// Mitsubishi GX Works2 project: Group27   PLC: FX3G

// global labels: Global1
VAR_GLOBAL
  Start_Day AT X007 : BOOL;
  Input_Raspberry AT D1100 : INT;
  Raspberry AT D1200 : INT;
  Input_Lemon AT D1300 : INT;
  Lemon AT D1400 : INT;
  Input_Stabilizer AT D1500 : INT;
  Stabilizer AT D1600 : INT;
  Input_Gummybears AT D1700 : INT;
  Gummybears AT D1800 : INT;
  Analog_Output2 AT D2500 : INT;
  Choice AT D1900 : REAL;
  Raspberry_Icecream_Container AT D2000 : INT;
  Lemon_Icecream_Cointainer AT D2100 : INT;
  Analog_Input1 AT D8280 : INT;
  Raspberry_Icecream_Cooler AT D2200 : INT;
  Lemon_Icecream_Cooler AT D2300 : INT;
  Mixing_Container AT D2400 : INT;
  Not_Enough_Material AT M1 : BOOL;
  Normal_Lamp AT M2 : BOOL;
  Pinuk_Lamp AT M3 : BOOL;
  Finished_Move_Cool AT M4 : BOOL;
  Cool_Finished AT M5 : BOOL;
  Trigger_Blink AT M6 : BOOL;
  Finish_Work AT M7 : BOOL;
  Zero AT K0 : INT;
  In_Work AT Y007 : BOOL;
  Emergency_Switch AT X005 : BOOL;
  Sample AT X001 : BOOL;
  Analog_Output AT D8282 : INT;
  Divider_400 AT E400 : REAL;
  Max_Normal AT E5 : REAL;
  Min_Pinuk AT E5 : REAL;
  Min_Raspberry_Normal AT K280 : INT;
  Min_Raspberry_Pinuk AT K385 : INT;
  Min_Lemon_Normal AT K455 : INT;
  Min_Lemon_Pinuk AT K665 : INT;
  Min_Stabilizer_Normal AT K105 : INT;
  Min_Stabilizer_Pinuk AT K210 : INT;
  Min_Gummybear_Normal AT K28 : INT;
  Min_Gummybear_Pinuk AT K70 : INT;
  Raspberry_Icecream_Normal AT K350 : INT;
  Raspberry_Icecream_Pinuk AT K560 : INT;
  Lemon_Icecream_Normal AT K490 : INT;
  Lemon_Icecream_Pinuk AT K700 : INT;
  Add_Pack AT K1 : INT;
  One_Sec AT K10 : INT;
  Three_Sec AT K30 : INT;
  Five_Sec AT K50 : INT;
  Eight_Sec AT K80 : INT;
  Normal_Icecram AT K868 : INT;
  Pinuk_Icecram AT K1330 : INT;
  Multiply_40 AT K40 : INT;
  First_Step_Timer AT TC0 : BOOL;
  Step1_Finished AT TS0 : BOOL;
  Icecream_Making AT Y000 : BOOL;
  Start_Cool AT X002 : BOOL;
  Second_Step_Timer AT TC1 : BOOL;
  Step2_Finished AT TS1 : BOOL;
  Temp10 AT X003 : BOOL;
  During_Cool AT Y002 : BOOL;
  Timer_Blink1 AT TC3 : BOOL;
  Timer_Blink1_Finished AT TS3 : BOOL;
  Flash_Lamp1 AT Y005 : BOOL;
  Timer_Blink2 AT TC4 : BOOL;
  Timer_Blink2_Finished AT TS4 : BOOL;
  Flash_Lamp2 AT Y006 : BOOL;
  Third_Step_Timer_Pinuk AT TC5 : BOOL;
  Third_Step_Timer_Normal AT TC2 : BOOL;
  Step3_Finished_Normal AT TS2 : BOOL;
  Step3_Finished_Pinuk AT TS5 : BOOL;
END_VAR

// task Task_01 (event TRUE, interval 0, priority 31): POU_01

PROGRAM POU_01
(* structured ladder/FBD written out as ST: instructions are called as NAME(EN, inputs, outputs); _pN, _eN, _tN stand for wires *)
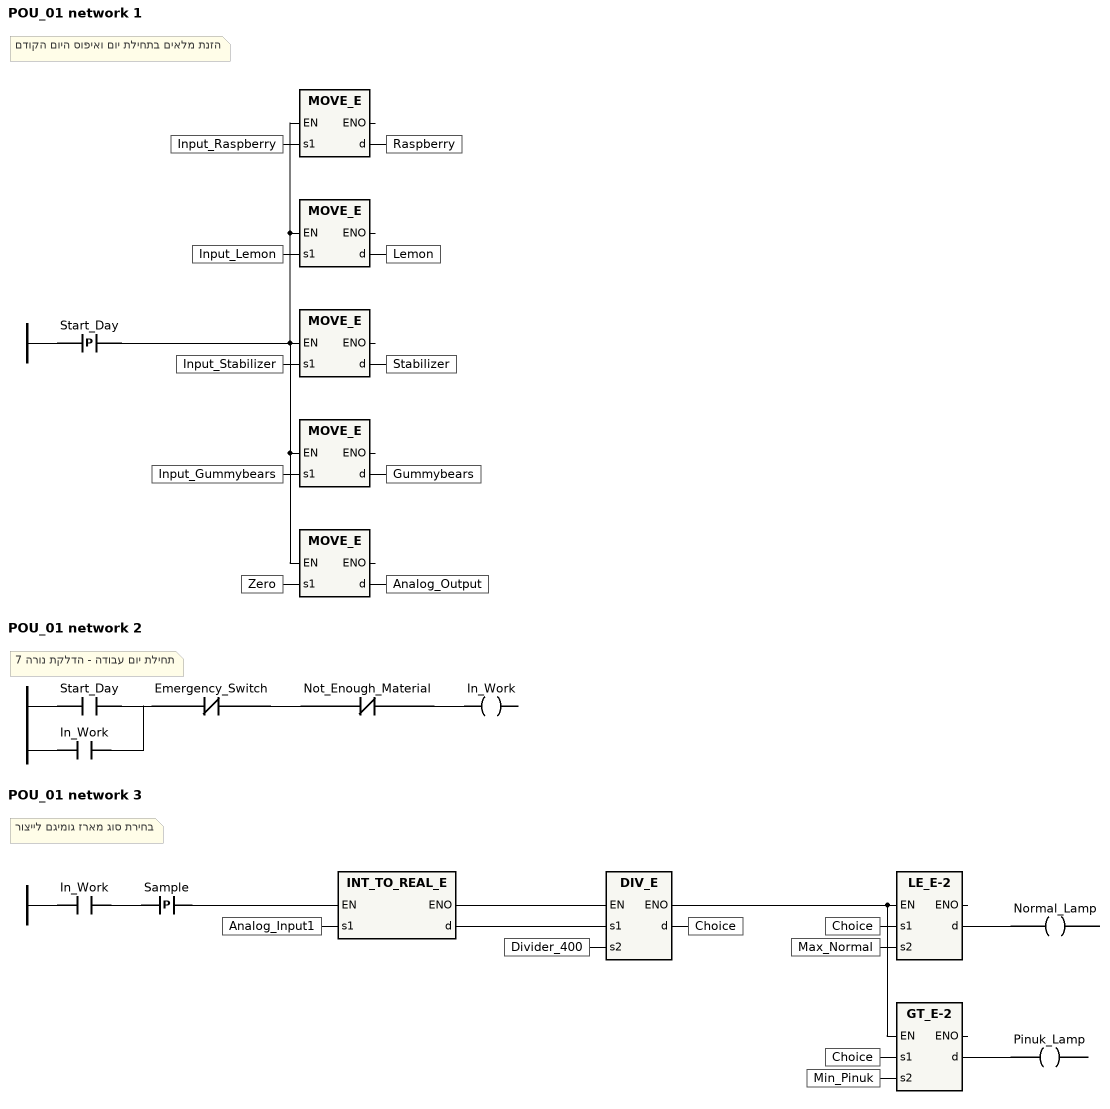
(* network 1 *)
(* הזנת מלאים בתחילת יום ואיפוס היום הקודם *)
_p1 := LDP(TRUE, Start_Day);
MOVE_E(_p1, Input_Raspberry, Raspberry);
MOVE_E(_p1, Input_Lemon, Lemon);
MOVE_E(_p1, Input_Stabilizer, Stabilizer);
MOVE_E(_p1, Input_Gummybears, Gummybears);
MOVE_E(_p1, Zero, Analog_Output);
(* network 2 *)
(* תחילת יום עבודה - הדלקת נורה 7 *)
In_Work := ((Start_Day OR In_Work) AND NOT Emergency_Switch) AND NOT Not_Enough_Material;
(* network 3 *)
(* בחירת סוג מארז גומיגם לייצור *)
_e2 := INT_TO_REAL_E(In_Work AND LDP(TRUE, Sample), Analog_Input1, _t1);
_e3 := DIV_E(_e2, _t1, Divider_400, Choice);
LE_E(_e3, Choice, Max_Normal, _t4);
Normal_Lamp := _t4;
GT_E(_e3, Choice, Min_Pinuk, _t5);
Pinuk_Lamp := _t5;
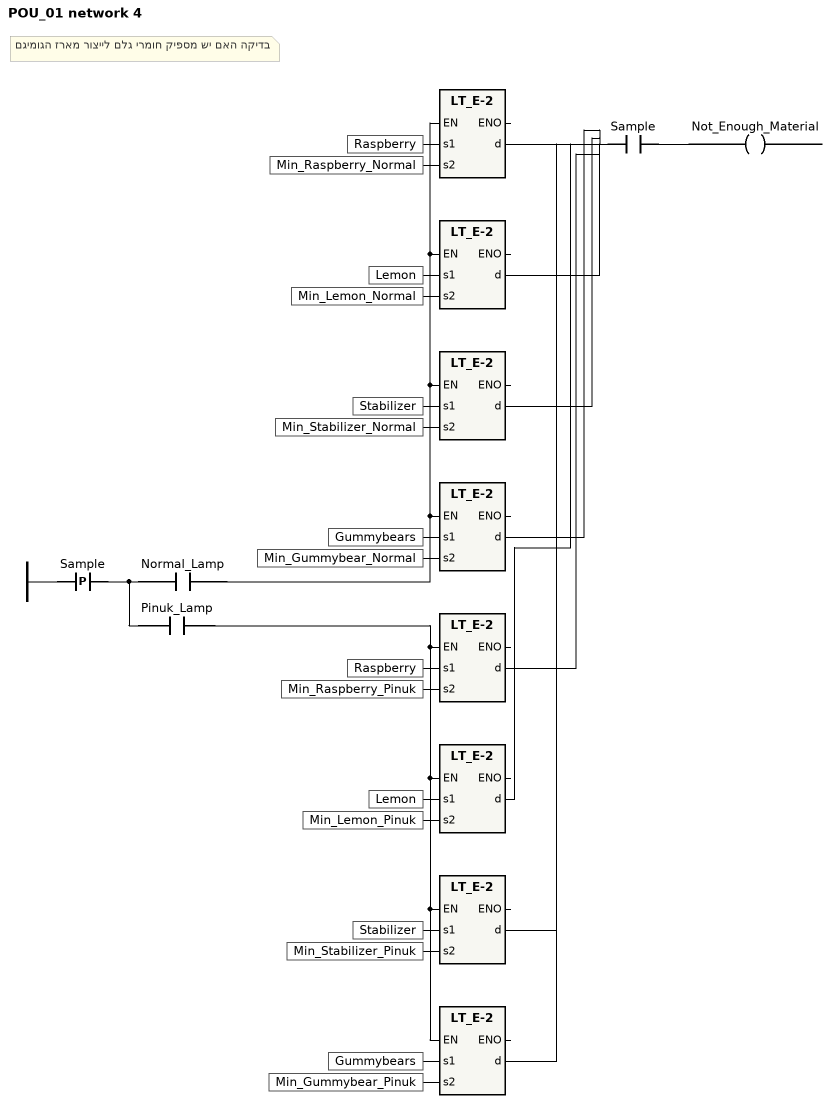
(* network 4 *)
(* בדיקה האם יש מספיק חומרי גלם לייצור מארז הגומיגם *)
_p1 := LDP(TRUE, Sample);
_p2 := _p1 AND Normal_Lamp;
LT_E(_p2, Raspberry, Min_Raspberry_Normal, _t3);
LT_E(_p2, Lemon, Min_Lemon_Normal, _t4);
LT_E(_p2, Stabilizer, Min_Stabilizer_Normal, _t5);
LT_E(_p2, Gummybears, Min_Gummybear_Normal, _t6);
_p7 := _p1 AND Pinuk_Lamp;
LT_E(_p7, Raspberry, Min_Raspberry_Pinuk, _t8);
LT_E(_p7, Lemon, Min_Lemon_Pinuk, _t9);
LT_E(_p7, Stabilizer, Min_Stabilizer_Pinuk, _t10);
LT_E(_p7, Gummybears, Min_Gummybear_Pinuk, _t11);
Not_Enough_Material := (_t3 OR _t4 OR _t5 OR _t6 OR _t8 OR _t9 OR _t10 OR _t11) AND Sample;
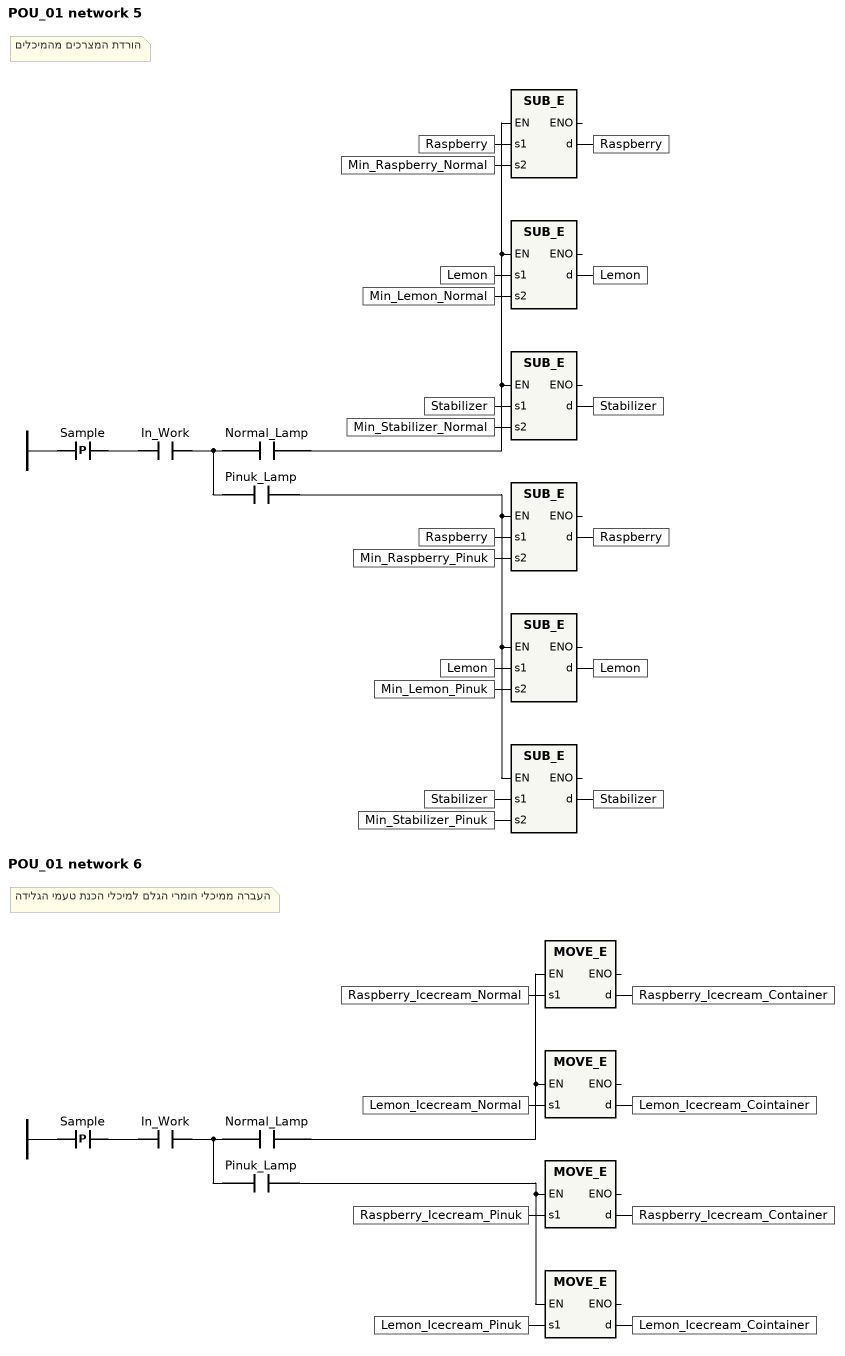
(* network 5 *)
(* הורדת המצרכים מהמיכלים *)
_p1 := LDP(TRUE, Sample) AND In_Work;
_p2 := _p1 AND Normal_Lamp;
SUB_E(_p2, Raspberry, Min_Raspberry_Normal, Raspberry);
SUB_E(_p2, Lemon, Min_Lemon_Normal, Lemon);
SUB_E(_p2, Stabilizer, Min_Stabilizer_Normal, Stabilizer);
_p3 := _p1 AND Pinuk_Lamp;
SUB_E(_p3, Raspberry, Min_Raspberry_Pinuk, Raspberry);
SUB_E(_p3, Lemon, Min_Lemon_Pinuk, Lemon);
SUB_E(_p3, Stabilizer, Min_Stabilizer_Pinuk, Stabilizer);
(* network 6 *)
(* העברה ממיכלי חומרי הגלם למיכלי הכנת טעמי הגלידה *)
_p1 := LDP(TRUE, Sample) AND In_Work;
_p2 := _p1 AND Normal_Lamp;
MOVE_E(_p2, Raspberry_Icecream_Normal, Raspberry_Icecream_Container);
MOVE_E(_p2, Lemon_Icecream_Normal, Lemon_Icecream_Cointainer);
_p3 := _p1 AND Pinuk_Lamp;
MOVE_E(_p3, Raspberry_Icecream_Pinuk, Raspberry_Icecream_Container);
MOVE_E(_p3, Lemon_Icecream_Pinuk, Lemon_Icecream_Cointainer);
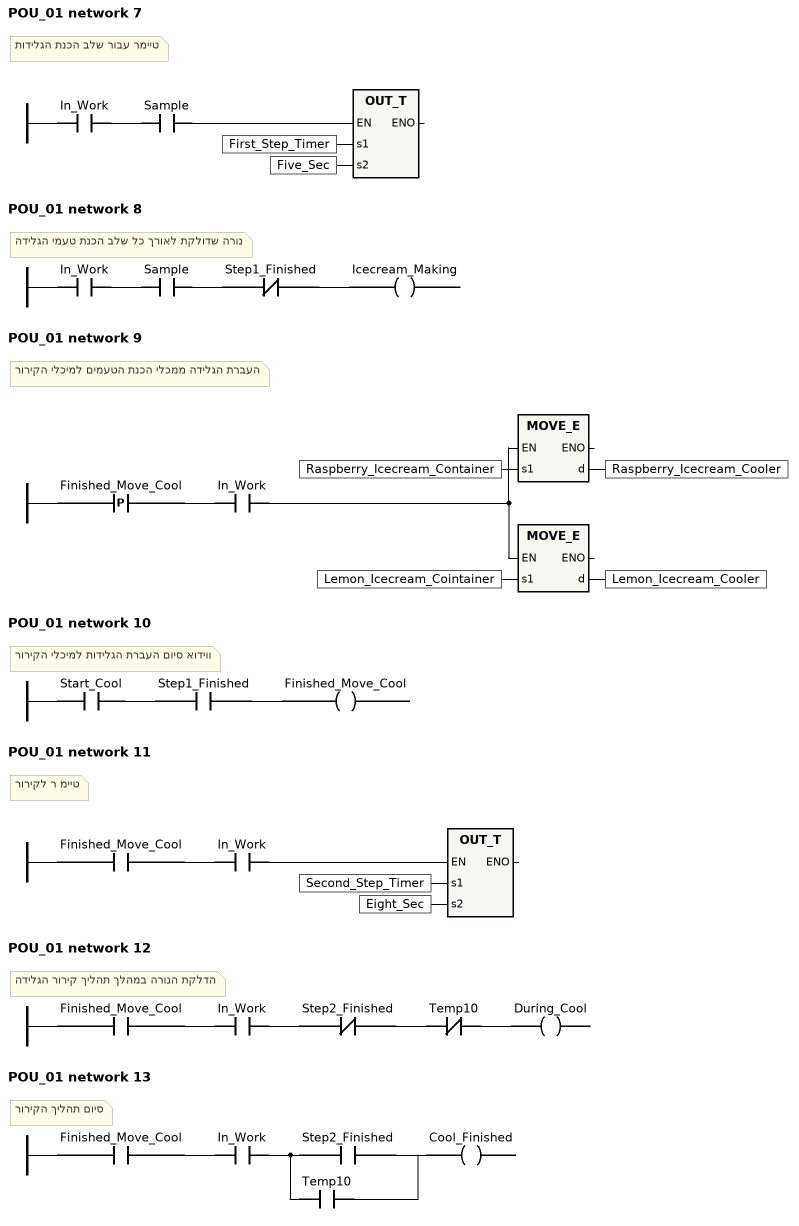
(* network 7 *)
(* טיימר עבור שלב הכנת הגלידות *)
OUT_T(In_Work AND Sample, First_Step_Timer, Five_Sec);
(* network 8 *)
(* נורה שדולקת לאורך כל שלב הכנת טעמי הגלידה *)
Icecream_Making := In_Work AND Sample AND NOT Step1_Finished;
(* network 9 *)
(* העברת הגלידה ממכלי הכנת הטעמים למיכלי הקירור *)
_p1 := LDP(TRUE, Finished_Move_Cool) AND In_Work;
MOVE_E(_p1, Raspberry_Icecream_Container, Raspberry_Icecream_Cooler);
MOVE_E(_p1, Lemon_Icecream_Cointainer, Lemon_Icecream_Cooler);
(* network 10 *)
(* ווידוא סיום העברת הגלידות למיכלי הקירור *)
Finished_Move_Cool := Start_Cool AND Step1_Finished;
(* network 11 *)
(* טיימ ר לקירור *)
OUT_T(Finished_Move_Cool AND In_Work, Second_Step_Timer, Eight_Sec);
(* network 12 *)
(* הדלקת הנורה במהלך תהליך קירור הגלידה *)
During_Cool := Finished_Move_Cool AND In_Work AND NOT Step2_Finished AND NOT Temp10;
(* network 13 *)
(* סיום תהליך הקירור *)
_p1 := Finished_Move_Cool AND In_Work;
Cool_Finished := (_p1 AND Step2_Finished) OR (_p1 AND Temp10);
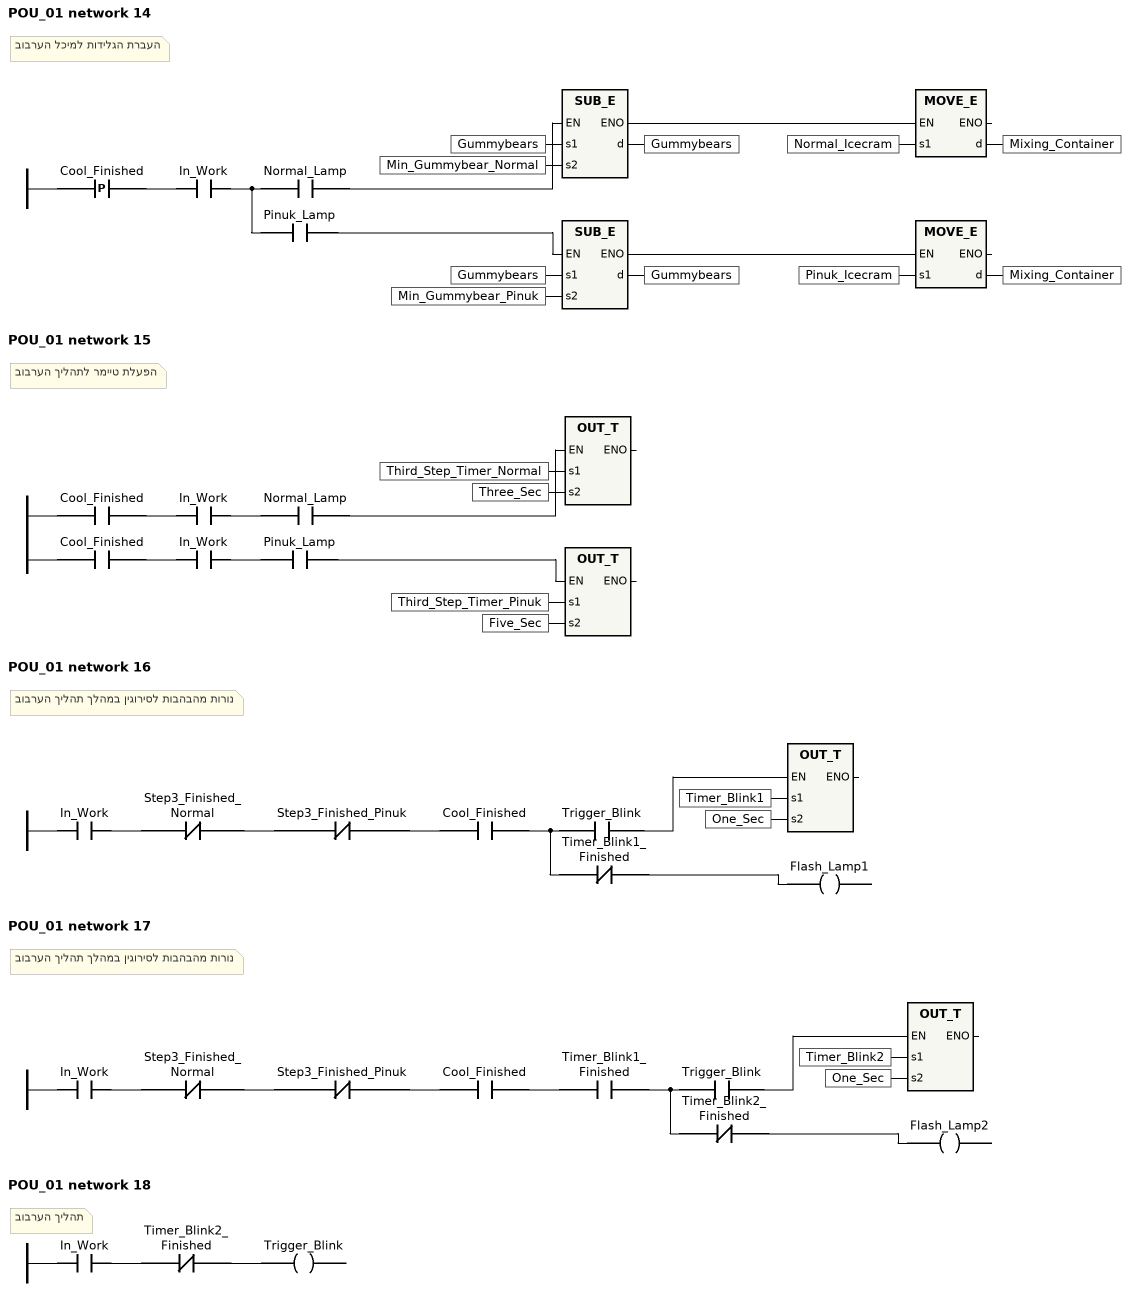
(* network 14 *)
(* העברת הגלידות למיכל הערבוב *)
_p1 := LDP(TRUE, Cool_Finished) AND In_Work;
_e2 := SUB_E(_p1 AND Normal_Lamp, Gummybears, Min_Gummybear_Normal, Gummybears);
MOVE_E(_e2, Normal_Icecram, Mixing_Container);
_e3 := SUB_E(_p1 AND Pinuk_Lamp, Gummybears, Min_Gummybear_Pinuk, Gummybears);
MOVE_E(_e3, Pinuk_Icecram, Mixing_Container);
(* network 15 *)
(* הפעלת טיימר לתהליך הערבוב *)
OUT_T(Cool_Finished AND In_Work AND Normal_Lamp, Third_Step_Timer_Normal, Three_Sec);
OUT_T(Cool_Finished AND In_Work AND Pinuk_Lamp, Third_Step_Timer_Pinuk, Five_Sec);
(* network 16 *)
(* נורות מהבהבות לסירוגין במהלך תהליך הערבוב *)
_p1 := In_Work AND NOT Step3_Finished_Normal AND NOT Step3_Finished_Pinuk AND Cool_Finished;
OUT_T(_p1 AND Trigger_Blink, Timer_Blink1, One_Sec);
Flash_Lamp1 := _p1 AND NOT Timer_Blink1_Finished;
(* network 17 *)
(* נורות מהבהבות לסירוגין במהלך תהליך הערבוב *)
_p1 := In_Work AND NOT Step3_Finished_Normal AND NOT Step3_Finished_Pinuk AND Cool_Finished AND Timer_Blink1_Finished;
OUT_T(_p1 AND Trigger_Blink, Timer_Blink2, One_Sec);
Flash_Lamp2 := _p1 AND NOT Timer_Blink2_Finished;
(* network 18 *)
(* תהליך הערבוב *)
Trigger_Blink := In_Work AND NOT Timer_Blink2_Finished;
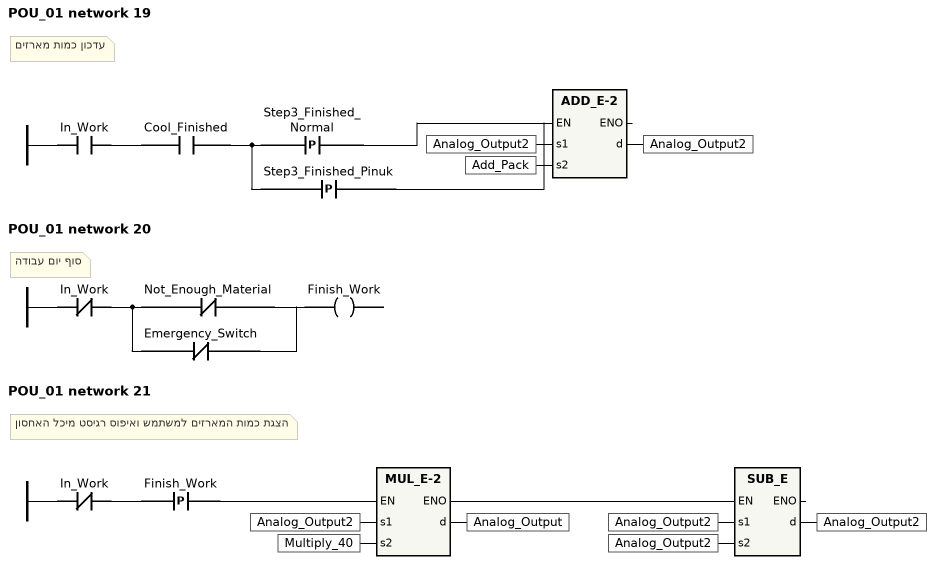
(* network 19 *)
(* עדכון כמות מארזים *)
_p1 := In_Work AND Cool_Finished;
ADD_E((_p1 AND LDP(TRUE, Step3_Finished_Normal)) OR (_p1 AND LDP(TRUE, Step3_Finished_Pinuk)), Analog_Output2, Add_Pack, Analog_Output2);
(* network 20 *)
(* סוף יום עבודה *)
_p1 := NOT In_Work;
Finish_Work := (_p1 AND NOT Not_Enough_Material) OR (_p1 AND NOT Emergency_Switch);
(* network 21 *)
(* הצגת כמות המארזים למשתמש ואיפוס רגיסט מיכל האחסון *)
_e1 := MUL_E(NOT In_Work AND LDP(TRUE, Finish_Work), Analog_Output2, Multiply_40, Analog_Output);
SUB_E(_e1, Analog_Output2, Analog_Output2, Analog_Output2);
END_PROGRAM
